// Mitsubishi GX Works2 project: 240430_timechart1   PLC: Q03UDV

PROGRAM MAIN
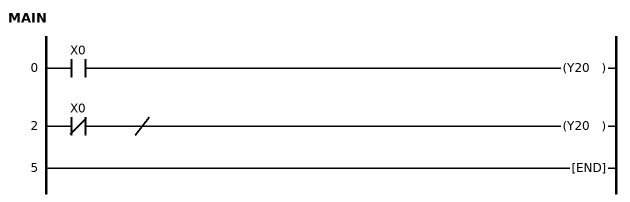
0     LD      X0
      OUT     Y20
2     LDI     X0
      INV
      OUT     Y20
5     END
END_PROGRAM
